(* PLC project Unnamed, Unknown Unnamed 1 *)
(* stored: creationDateTime 2025-06-20T21:12:14, modificationDateTime 2025-06-20T21:21:49 *)

PROGRAM bitwise
  VAR
    input1 AT %IX100.0 : BOOL;
    input2 AT %IX100.1 : BOOL;
    reset AT %IX100.2 : BOOL;
    load AT %IX100.3 : BOOL;
    output1 AT %QX100.0 : BOOL;
  END_VAR

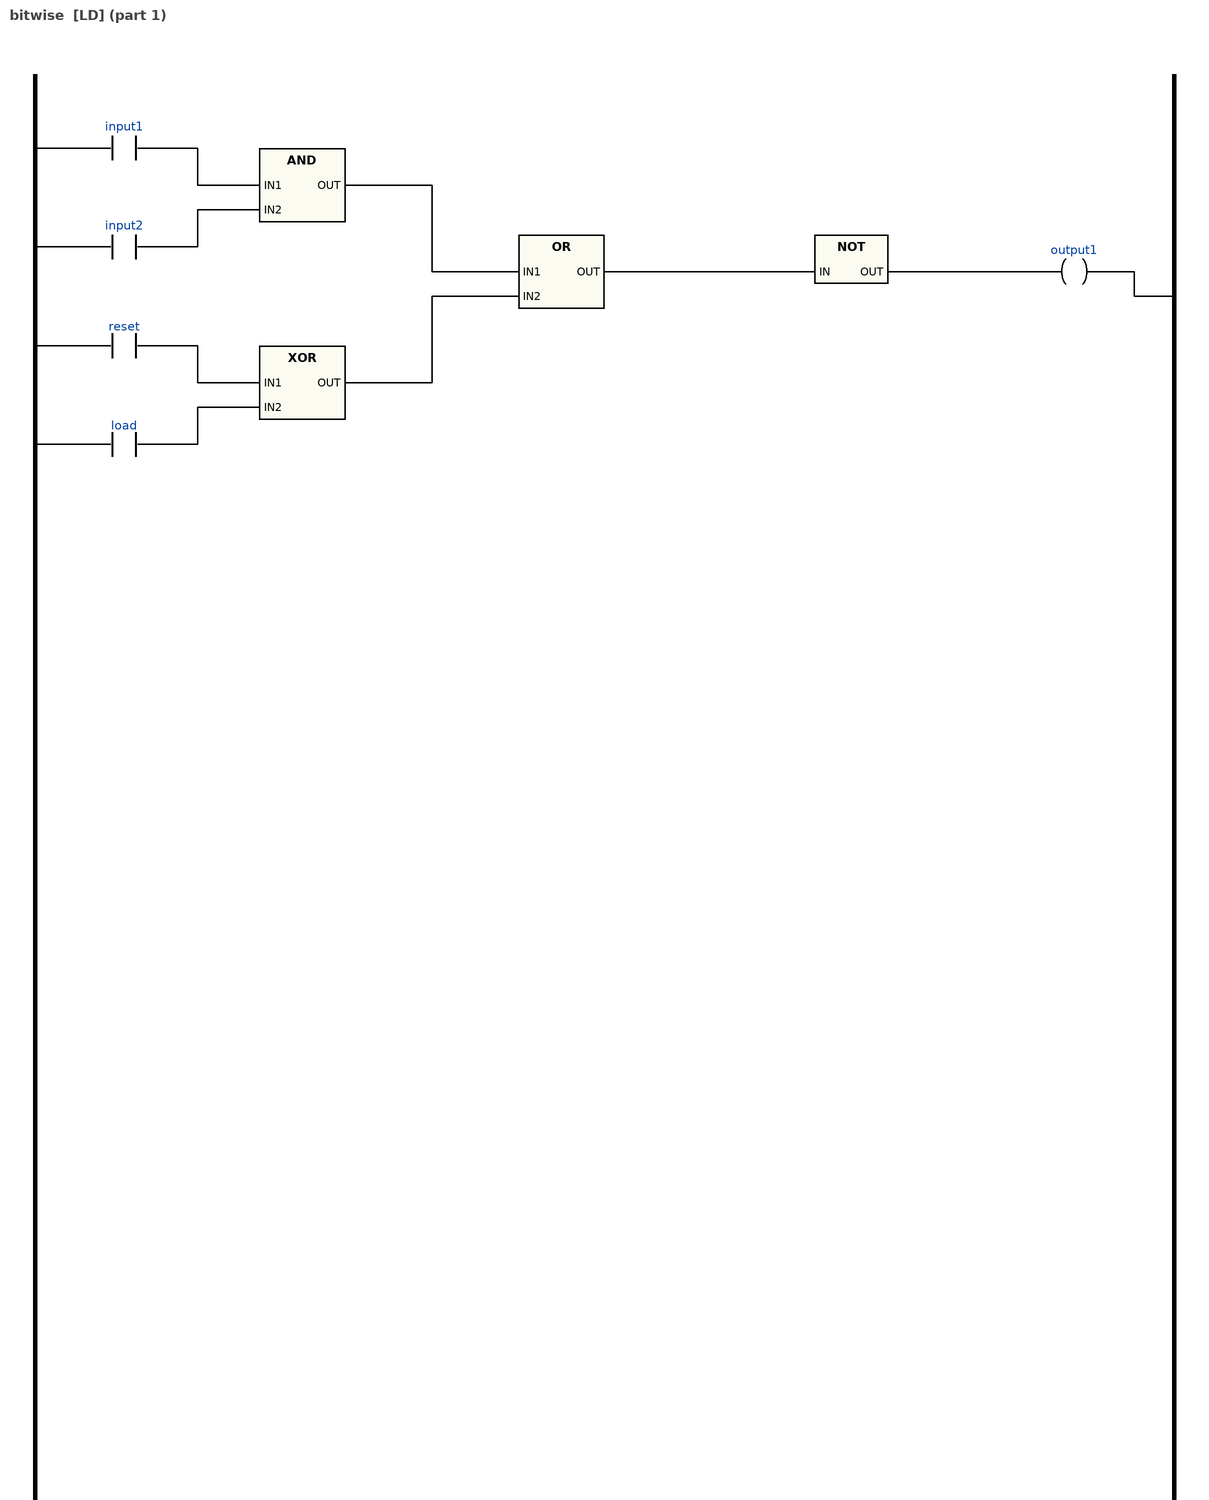
(* LD diagram, written out as Structured Text *)
output1 := NOT (input1 AND input2 OR reset XOR load);
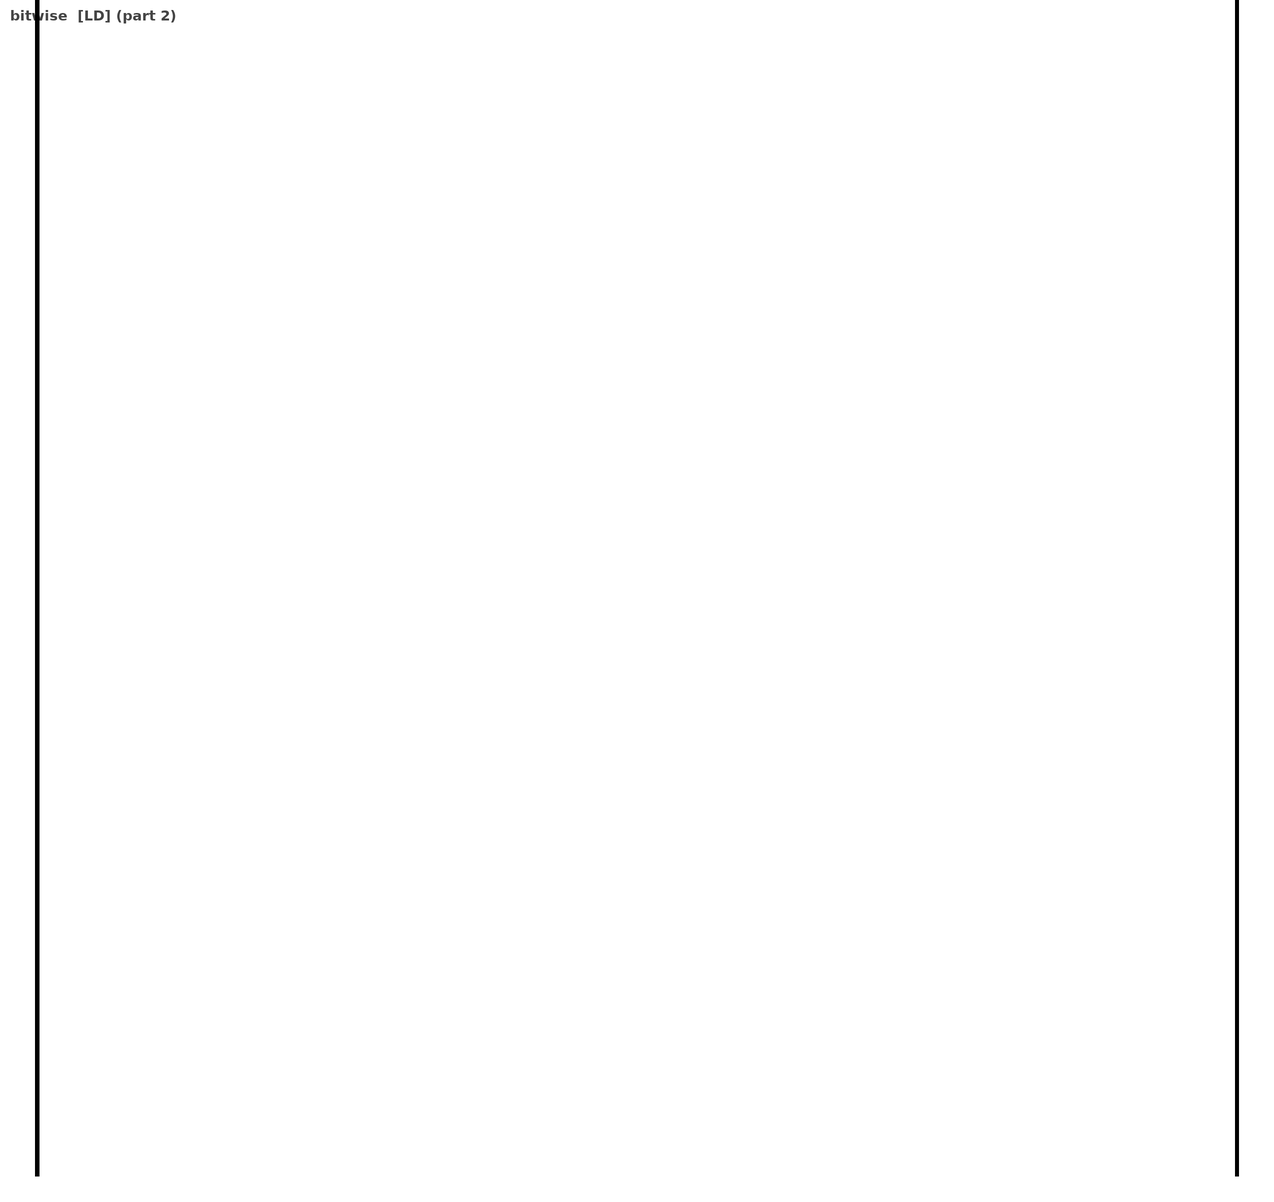
END_PROGRAM

CONFIGURATION Config0
  RESOURCE Res0 ON PLC
    TASK task0(INTERVAL := T#20ms, PRIORITY := 0);
    PROGRAM instance0 WITH task0 : bitwise;
  END_RESOURCE
END_CONFIGURATION
